(* PLC project Tc2_Utilities.FB_SetTimeZoneInformation Demo, tc3-libraries-kb TwinCAT 3.1 *)
(* stored: creationDateTime 2026-05-11T00:00:00, modificationDateTime 2026-05-11T00:00:00 *)

PROGRAM P_Demo_FB_SetTimeZoneInformation
  VAR
    fbFB_SetTimeZoneInformation : FB_SetTimeZoneInformation;  (* FB_SetTimeZoneInformation 实例 *)
    bWrite : BOOL := FALSE;
    stTzToSet : TIME_ZONE_INFORMATION;
    bBusy_ : BOOL;
    bErrFlag : BOOL;
    nErrCode : UDINT;
  END_VAR

// =============================================================================
// 场景：commissioning 时把所有机器时区统一改成 CST。
// 价值：替代手工进控制面板。
// 验证：先用 FB_GetTimeZoneInformation 读旧时区；触发写入新时区；再读应已切换。
// 验证步骤：
//   1. 右键 PLC 项目 → Import PLCopenXML → 选本文件
//   2. 引用 Tc2_Utilities（References → Add library）
//   3. 编译 → 登录 → 运行；按上方『验证』行的指示在线写值观察
// =============================================================================

fbFB_SetTimeZoneInformation(
    sNetID := '', bExecute := bWrite, tzInfo := stTzToSet, tTimeout := DEFAULT_ADS_TIMEOUT,
    bBusy => bBusy_, bErr => bErrFlag, nErrId => nErrCode
);
END_PROGRAM
